FUNCTION_BLOCK MUX_COLOR (* See MUX_ANY *)
  (* Standard: 61131-3 *)
  (* Version 0.0, 2004-12-15, JHC, Rockwell Automation, Converted from SRC format. *)
  (* Compiler header: package fb.rt.plc.select; *)
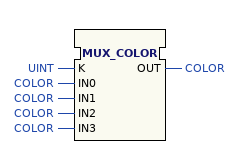
  VAR_INPUT
    K : UINT;
    IN0 : COLOR;
    IN1 : COLOR;
    IN2 : COLOR;
    IN3 : COLOR;
  END_VAR
  VAR_OUTPUT
    OUT : COLOR;
  END_VAR
END_FUNCTION_BLOCK
